FUNCTION fun_setAlarm : bool
VAR_INPUT
	in_flg_set : BOOL;
	in_flg_reset : BOOL;
END_VAR
VAR

END_VAR


	IF in_flg_reset = FALSE THEN
		IF in_flg_set THEN
			fun_setAlarm := TRUE;
		END_IF
	ELSIF in_flg_reset THEN
		fun_setAlarm := FALSE;
	END_IF

END_FUNCTION

(* stored: Version 1.1.0.1, ProductVersion 3.1.4024.11
   POU fun_setAlarm: Id {eeeb4bee-4d62-400d-ba48-5ded1f80b27c}, SpecialFunc None *)
